(* IEC 61131-3 sources: greenbuddies-ems-concept/docs/data-model/codesys, 10 files *)

(* ---- EmsReference.st ---- *)
(* GENERATED by npm run model:generate. Create one DUT for each TYPE block. *)

TYPE ST_EmsMeta :
STRUCT
    Quality : USINT := 6; (* 0=good, 1=uncertain, 2=bad, 3=stale, 4=unsupported, 5=disabled, 6=initializing *)
    ObservedAtMs : ULINT; (* UTC Unix ms; 0 means unknown in this PLC adapter *)
    Sequence : UDINT; (* Per-point successful observation counter; wraps to 1 *)
END_STRUCT
END_TYPE

TYPE ST_EmsNumber :
STRUCT
    Value : LREAL;
    Meta : ST_EmsMeta;
END_STRUCT
END_TYPE

TYPE ST_EmsBoolean :
STRUCT
    Value : BOOL;
    Meta : ST_EmsMeta;
END_STRUCT
END_TYPE

TYPE ST_EmsText :
STRUCT
    Value : STRING(255);
    Meta : ST_EmsMeta;
END_STRUCT
END_TYPE

TYPE ST_EmsCounter :
STRUCT
    Value : ULINT;
    Meta : ST_EmsMeta;
END_STRUCT
END_TYPE

TYPE ST_EmsDecoded :
STRUCT
    Value : LREAL;
    Valid : BOOL;
END_STRUCT
END_TYPE

TYPE U_EmsReal32 :
UNION
    Bits : DWORD;
    Value : REAL;
END_UNION
END_TYPE

TYPE ST_EmsDevice :
STRUCT
    online : ST_EmsBoolean; (* device.online | state | r | Last device transaction succeeded; does not imply every point is healthy. *)
    state : ST_EmsText; (* device.state | state | r | Normalized operating state; unknown codes map to unknown, never running. *)
    available : ST_EmsBoolean; (* device.available | state | r | Device reports available for operation. *)
    remoteMode : ST_EmsBoolean; (* device.remoteMode | state | r | Device accepts remote control at its own interface. *)
    faultActive : ST_EmsBoolean; (* device.faultActive | state | r | At least one device fault is active. *)
    warningActive : ST_EmsBoolean; (* device.warningActive | state | r | At least one device warning is active. *)
    vendorCode : ST_EmsText; (* device.vendorCode | state | r | Unmodified diagnostic code for service; never drives portable UI behavior. *)
    latency : ST_EmsNumber; (* device.latency | ms | r | Most recent successful transaction duration. *)
    uptime : ST_EmsCounter; (* device.uptime | s | r | Device uptime. A reset is not negative consumption. *)
    communicationErrors : ST_EmsCounter; (* device.communicationErrors | count | r | Cumulative failed transactions since source restart. *)
END_STRUCT
END_TYPE

TYPE ST_EmsAc :
STRUCT
    activePower : ST_EmsNumber; (* ac.activePower | W | r | Signed active power at the declared measurement boundary. *)
    reactivePower : ST_EmsNumber; (* ac.reactivePower | var | r | Signed reactive power at the same boundary as activePower. *)
    apparentPower : ST_EmsNumber; (* ac.apparentPower | VA | r | Non-negative apparent power. *)
    frequency : ST_EmsNumber; (* ac.frequency | Hz | r | Measured AC frequency. *)
    powerFactor : ST_EmsNumber; (* ac.powerFactor | 1 | r | P / apparent power, signed by active power; null if undefined. *)
    voltageL1N : ST_EmsNumber; (* ac.voltageL1N | V | r | L1 to neutral RMS voltage. *)
    voltageL2N : ST_EmsNumber; (* ac.voltageL2N | V | r | L2 to neutral RMS voltage. *)
    voltageL3N : ST_EmsNumber; (* ac.voltageL3N | V | r | L3 to neutral RMS voltage. *)
    voltageL1L2 : ST_EmsNumber; (* ac.voltageL1L2 | V | r | L1 to L2 RMS voltage. *)
    voltageL2L3 : ST_EmsNumber; (* ac.voltageL2L3 | V | r | L2 to L3 RMS voltage. *)
    voltageL3L1 : ST_EmsNumber; (* ac.voltageL3L1 | V | r | L3 to L1 RMS voltage. *)
    currentL1 : ST_EmsNumber; (* ac.currentL1 | A | r | L1 RMS current magnitude. *)
    currentL2 : ST_EmsNumber; (* ac.currentL2 | A | r | L2 RMS current magnitude. *)
    currentL3 : ST_EmsNumber; (* ac.currentL3 | A | r | L3 RMS current magnitude. *)
    activePowerL1 : ST_EmsNumber; (* ac.activePowerL1 | W | r | Signed active power, L1. *)
    activePowerL2 : ST_EmsNumber; (* ac.activePowerL2 | W | r | Signed active power, L2. *)
    activePowerL3 : ST_EmsNumber; (* ac.activePowerL3 | W | r | Signed active power, L3. *)
    voltageThd : ST_EmsNumber; (* ac.voltageThd | % | r | Reported aggregate voltage total harmonic distortion. *)
END_STRUCT
END_TYPE

TYPE ST_EmsDc :
STRUCT
    voltage : ST_EmsNumber; (* dc.voltage | V | r | DC terminal voltage. *)
    current : ST_EmsNumber; (* dc.current | A | r | DC current; positive out of the asset. *)
    power : ST_EmsNumber; (* dc.power | W | r | DC power; positive out of the asset. *)
    insulationResistance : ST_EmsNumber; (* dc.insulationResistance | ohm | r | Insulation resistance to ground. *)
END_STRUCT
END_TYPE

TYPE ST_EmsEnergy :
STRUCT
    exported : ST_EmsCounter; (* energy.exported | Wh | r | Cumulative active energy leaving the boundary. *)
    imported : ST_EmsCounter; (* energy.imported | Wh | r | Cumulative active energy entering the boundary. *)
    generatedToday : ST_EmsNumber; (* energy.generatedToday | Wh | r | Generation since site-local midnight; date/timezone are metadata. *)
    exportedToday : ST_EmsNumber; (* energy.exportedToday | Wh | r | Export since site-local midnight. *)
    importedToday : ST_EmsNumber; (* energy.importedToday | Wh | r | Import since site-local midnight. *)
    runtime : ST_EmsCounter; (* energy.runtime | s | r | Cumulative operating time. *)
END_STRUCT
END_TYPE

TYPE ST_EmsPv :
STRUCT
    moduleTemperature : ST_EmsNumber; (* pv.moduleTemperature | degC | r | PV module temperature. *)
    inverterTemperature : ST_EmsNumber; (* pv.inverterTemperature | degC | r | Inverter internal temperature. *)
    irradiance : ST_EmsNumber; (* pv.irradiance | W/m2 | r | Plane-of-array irradiance. *)
    availablePower : ST_EmsNumber; (* pv.availablePower | W | r | Device-estimated available active power; not inferred from nameplate. *)
    curtailedPower : ST_EmsNumber; (* pv.curtailedPower | W | r | Reported curtailed active power. *)
END_STRUCT
END_TYPE

TYPE ST_EmsBattery :
STRUCT
    soc : ST_EmsNumber; (* battery.soc | % | r | State of charge. *)
    soh : ST_EmsNumber; (* battery.soh | % | r | State of health. *)
    storedEnergy : ST_EmsNumber; (* battery.storedEnergy | Wh | r | Estimated stored usable energy. *)
    chargeAvailable : ST_EmsNumber; (* battery.chargeAvailable | W | r | Maximum currently available charge magnitude. *)
    dischargeAvailable : ST_EmsNumber; (* battery.dischargeAvailable | W | r | Maximum currently available discharge magnitude. *)
    temperature : ST_EmsNumber; (* battery.temperature | degC | r | Reported representative battery temperature. *)
    minTemperature : ST_EmsNumber; (* battery.minTemperature | degC | r | Lowest measured temperature. *)
    maxTemperature : ST_EmsNumber; (* battery.maxTemperature | degC | r | Highest measured temperature. *)
    minCellVoltage : ST_EmsNumber; (* battery.minCellVoltage | V | r | Lowest measured cell voltage. *)
    maxCellVoltage : ST_EmsNumber; (* battery.maxCellVoltage | V | r | Highest measured cell voltage. *)
    cycles : ST_EmsCounter; (* battery.cycles | count | r | Completed equivalent cycles; fractional cycles require a separate extension field. *)
    contactorClosed : ST_EmsBoolean; (* battery.contactorClosed | state | r | Battery contactor closed readback. *)
    balancing : ST_EmsBoolean; (* battery.balancing | state | r | Cell balancing active. *)
END_STRUCT
END_TYPE

TYPE ST_EmsWind :
STRUCT
    speed : ST_EmsNumber; (* wind.speed | m/s | r | Wind speed at the instrument. *)
    direction : ST_EmsNumber; (* wind.direction | deg | r | Wind direction, clockwise from true north. *)
    rotorSpeed : ST_EmsNumber; (* wind.rotorSpeed | rpm | r | Rotor speed. *)
    nacelleDirection : ST_EmsNumber; (* wind.nacelleDirection | deg | r | Nacelle bearing from true north. *)
    pitch : ST_EmsNumber; (* wind.pitch | deg | r | Reported representative blade pitch. *)
    gearboxTemperature : ST_EmsNumber; (* wind.gearboxTemperature | degC | r | Gearbox temperature. *)
    availablePower : ST_EmsNumber; (* wind.availablePower | W | r | Reported available generation. *)
END_STRUCT
END_TYPE

TYPE ST_EmsHydro :
STRUCT
    flow : ST_EmsNumber; (* hydro.flow | m3/s | r | Volumetric flow through the unit. *)
    head : ST_EmsNumber; (* hydro.head | m | r | Net hydraulic head. *)
    upstreamLevel : ST_EmsNumber; (* hydro.upstreamLevel | m | r | Upstream level relative to the configured datum. *)
    downstreamLevel : ST_EmsNumber; (* hydro.downstreamLevel | m | r | Downstream level relative to the same datum. *)
    gatePosition : ST_EmsNumber; (* hydro.gatePosition | % | r | Gate opening. *)
    turbineSpeed : ST_EmsNumber; (* hydro.turbineSpeed | rpm | r | Hydro turbine speed. *)
    waterTemperature : ST_EmsNumber; (* hydro.waterTemperature | degC | r | Water temperature. *)
END_STRUCT
END_TYPE

TYPE ST_EmsGrid :
STRUCT
    dsoAllowance : ST_EmsNumber; (* grid.dsoAllowance | % | r | Discrete DSO export allowance. *)
    exportLimit : ST_EmsNumber; (* grid.exportLimit | W | r | Effective non-negative export ceiling. *)
    importLimit : ST_EmsNumber; (* grid.importLimit | W | r | Effective non-negative import ceiling. *)
    connected : ST_EmsBoolean; (* grid.connected | state | r | PCC connected to the external grid. *)
    islanded : ST_EmsBoolean; (* grid.islanded | state | r | Site operating as an island. *)
    breakerClosed : ST_EmsBoolean; (* grid.breakerClosed | state | r | Breaker closed auxiliary-contact readback. *)
    tripActive : ST_EmsBoolean; (* grid.tripActive | state | r | Protection trip active. *)
    transformerTemperature : ST_EmsNumber; (* grid.transformerTemperature | degC | r | Transformer winding or oil sensor, identified in point metadata. *)
    tapPosition : ST_EmsNumber; (* grid.tapPosition | step | r | Transformer tap position; signed integral step. *)
END_STRUCT
END_TYPE

TYPE ST_EmsMeteo :
STRUCT
    airTemperature : ST_EmsNumber; (* meteo.airTemperature | degC | r | Ambient air temperature. *)
    humidity : ST_EmsNumber; (* meteo.humidity | % | r | Relative humidity. *)
    pressure : ST_EmsNumber; (* meteo.pressure | Pa | r | Atmospheric pressure. *)
    irradiance : ST_EmsNumber; (* meteo.irradiance | W/m2 | r | Global horizontal irradiance. *)
    windSpeed : ST_EmsNumber; (* meteo.windSpeed | m/s | r | Wind speed. *)
    windDirection : ST_EmsNumber; (* meteo.windDirection | deg | r | Direction clockwise from true north. *)
    rainfall : ST_EmsNumber; (* meteo.rainfall | mm | r | Precipitation in the configured measurement window. *)
END_STRUCT
END_TYPE

TYPE ST_EmsLoad :
STRUCT
    demand : ST_EmsNumber; (* load.demand | W | r | Non-negative active power consumed. *)
    flexiblePower : ST_EmsNumber; (* load.flexiblePower | W | r | Reported shed-able load magnitude. *)
    enabled : ST_EmsBoolean; (* load.enabled | state | r | Load enabled readback. *)
    vehicleConnected : ST_EmsBoolean; (* load.vehicleConnected | state | r | Vehicle present at this connector. *)
    charging : ST_EmsBoolean; (* load.charging | state | r | Charging active readback. *)
    currentLimit : ST_EmsNumber; (* load.currentLimit | A | r | Accepted EV connector current limit. *)
    sessionEnergy : ST_EmsNumber; (* load.sessionEnergy | Wh | r | Energy delivered in this charging session. *)
END_STRUCT
END_TYPE

TYPE ST_EmsController :
STRUCT
    mode : ST_EmsText; (* controller.mode | state | r | Current controller mode. *)
    source : ST_EmsText; (* controller.source | state | r | Exactly one selected command authority. *)
    remoteConnected : ST_EmsBoolean; (* controller.remoteConnected | state | r | Aggregator transport connected. *)
    remoteAllowed : ST_EmsBoolean; (* controller.remoteAllowed | state | rw | Remote permission readback; disabling selects local authority. *)
    requestedPower : ST_EmsNumber; (* controller.requestedPower | W | r | Requested aggregate active power before controller constraints. *)
    afterController : ST_EmsNumber; (* controller.afterController | W | r | Power after local optimization and device feasibility limits. *)
    afterDso : ST_EmsNumber; (* controller.afterDso | W | r | Power after DSO/export constraints. *)
    deliveredPower : ST_EmsNumber; (* controller.deliveredPower | W | r | Final dispatched power; distinct from measured power. *)
    limitingReason : ST_EmsText; (* controller.limitingReason | state | r | Dominant normalized active constraint. *)
END_STRUCT
END_TYPE

TYPE ST_EmsSettings :
STRUCT
    peakImportTarget : ST_EmsNumber; (* settings.peakImportTarget | W | rw | Peak-shaving import target. *)
    peakShavingShare : ST_EmsNumber; (* settings.peakShavingShare | % | rw | Usable battery allocation to peak shaving; remainder for load shifting. *)
    socMin : ST_EmsNumber; (* settings.socMin | % | rw | Minimum operating SoC; strictly below socMax. *)
    socMax : ST_EmsNumber; (* settings.socMax | % | rw | Maximum operating SoC; strictly above socMin. *)
    chargeLimit : ST_EmsNumber; (* settings.chargeLimit | W | rw | Requested maximum charge magnitude. *)
    dischargeLimit : ST_EmsNumber; (* settings.dischargeLimit | W | rw | Requested maximum discharge magnitude. *)
    rampLimit : ST_EmsNumber; (* settings.rampLimit | W/s | rw | Maximum change of active power magnitude per second. *)
END_STRUCT
END_TYPE

TYPE ST_EmsCamera :
STRUCT
    online : ST_EmsBoolean; (* camera.online | state | r | Camera reachable. *)
    recording : ST_EmsBoolean; (* camera.recording | state | r | Recording active. *)
    frameAge : ST_EmsNumber; (* camera.frameAge | ms | r | Age of most recently received image. *)
END_STRUCT
END_TYPE

TYPE ST_EmsAsset :
STRUCT
    Id : STRING(128);
    Kind : STRING(32);
    device : ST_EmsDevice;
    ac : ST_EmsAc;
    dc : ST_EmsDc;
    energy : ST_EmsEnergy;
    pv : ST_EmsPv;
    battery : ST_EmsBattery;
    wind : ST_EmsWind;
    hydro : ST_EmsHydro;
    grid : ST_EmsGrid;
    meteo : ST_EmsMeteo;
    load : ST_EmsLoad;
    controller : ST_EmsController;
    settings : ST_EmsSettings;
    camera : ST_EmsCamera;
END_STRUCT
END_TYPE

(* Additional DUTs. Fixed reference bounds: 64 intervals, 32 targets per interval. Reject larger input before copying. *)
TYPE ST_EmsTarget :
STRUCT
    AssetId : STRING(128);
    ActivePowerW : LREAL;
END_STRUCT
END_TYPE

TYPE ST_EmsInterval :
STRUCT
    StartMs : ULINT;
    EndMs : ULINT;
    TargetCount : UINT;
    Targets : ARRAY[1..32] OF ST_EmsTarget;
END_STRUCT
END_TYPE

TYPE ST_EmsProfile :
STRUCT
    Revision : STRING(128);
    ValidFromMs : ULINT;
    ValidUntilMs : ULINT;
    IntervalCount : UINT;
    Intervals : ARRAY[1..64] OF ST_EmsInterval;
END_STRUCT
END_TYPE

TYPE ST_EmsCommandResult :
STRUCT
    CommandId : STRING(128);
    Revision : STRING(128);
    State : STRING(32); (* received, validated, accepted, applied, rejected, expired *)
    Reason : STRING(255);
    AtMs : ULINT;
END_STRUCT
END_TYPE

(* ===== FB_EmsHighAlarm.st ===== *)
(* Create a FUNCTION_BLOCK POU. Declarations above, implementation below the divider.
   Requires the CODESYS Standard library (TON). Example settings are not safety limits.
   One instance per condition. Call every scan from ONE acquisition/alarm task.
   Acknowledgement belongs to Alarm Manager, never to this block. *)
FUNCTION_BLOCK FB_EmsHighAlarm
VAR_INPUT
    lrValue       : LREAL;
    xValid        : BOOL;        (* Good, fresh sample AND valid mapping *)
    lrHigh        : LREAL;
    lrReset       : LREAL;       (* Must be below lrHigh: hysteresis *)
    tRaiseDelay   : TIME := T#2s;
    tClearDelay   : TIME := T#5s;
END_VAR
VAR_OUTPUT
    xActive       : BOOL;        (* Digital alarm expression; never writable by HMI *)
    xInputFault   : BOOL;        (* Separate communication/measurement alarm *)
    xConfigFault  : BOOL;
END_VAR
VAR
    fbRaise       : TON;
    fbClear       : TON;
END_VAR
(* ---- Implementation ---- *)
xConfigFault := (lrReset >= lrHigh);
xInputFault := NOT xValid;
IF xInputFault OR xConfigFault THEN
    fbRaise(IN := FALSE, PT := tRaiseDelay);
    fbClear(IN := FALSE, PT := tClearDelay);
    (* Hold last known condition; unavailable data must not clear a fault. *)
ELSE
    fbRaise(IN := (NOT xActive) AND (lrValue >= lrHigh), PT := tRaiseDelay);
    fbClear(IN := xActive AND (lrValue <= lrReset), PT := tClearDelay);
    IF fbRaise.Q THEN
        xActive := TRUE;
    ELSIF fbClear.Q THEN
        xActive := FALSE;
    END_IF;
END_IF;
END_FUNCTION_BLOCK

(* ===== FB_EmsSample.st ===== *)
(* POU: FUNCTION_BLOCK FB_EmsSample. Declaration above the divider; implementation below it. *)
FUNCTION_BLOCK FB_EmsSample
VAR_INPUT
    xSupported : BOOL := TRUE;
    xEnabled : BOOL := TRUE;
    xNewSample : BOOL; (* One pulse per completed acquisition, NOT each PLC cycle. *)
    xReadError : BOOL; (* Failed transaction pulse; retained words are not new data. *)
    xValueValid : BOOL := TRUE;
    xClockValid : BOOL;
    uliUtcMs : ULINT;
    uliMonotonicMs : ULINT; (* LTIME_TO_ULINT(LTIME()) / ULINT#1000000 *)
    udiStaleAfterMs : UDINT := 5000;
END_VAR
VAR_OUTPUT
    Meta : ST_EmsMeta;
    xAccept : BOOL; (* Copy the decoded value only when TRUE. *)
END_VAR
VAR
    xSeen : BOOL;
    uliLastMs : ULINT;
END_VAR
(* IMPLEMENTATION *)
xAccept := FALSE;
IF NOT xSupported THEN
    Meta.Quality := 4; (* unsupported *)
    Meta.ObservedAtMs := 0;
    Meta.Sequence := 0;
    xSeen := FALSE;
ELSIF NOT xEnabled THEN
    Meta.Quality := 5; (* disabled; retain the last observation *)
ELSIF xReadError THEN
    Meta.Quality := 2; (* bad; preserve last observation time and value *)
ELSIF xNewSample THEN
    IF xValueValid THEN
        xAccept := TRUE;
        xSeen := TRUE;
        uliLastMs := uliMonotonicMs;
        IF xClockValid AND (uliUtcMs > 0) THEN
            Meta.Quality := 0;
            Meta.ObservedAtMs := uliUtcMs;
        ELSE
            Meta.Quality := 1; (* uncertain: no trustworthy UTC *)
            Meta.ObservedAtMs := 0;
        END_IF;
        IF Meta.Sequence = UDINT#4294967295 THEN
            Meta.Sequence := 1;
        ELSE
            Meta.Sequence := Meta.Sequence + 1;
        END_IF;
    ELSE
        Meta.Quality := 2; (* sentinel, range error or unmapped enum *)
    END_IF;
ELSIF xSeen THEN
    IF uliMonotonicMs < uliLastMs THEN
        Meta.Quality := 2; (* monotonic clock reset; wait for a new sample *)
    ELSIF (uliMonotonicMs - uliLastMs) > UDINT_TO_ULINT(udiStaleAfterMs) THEN
        Meta.Quality := 3; (* stale; UTC observation time stays unchanged *)
    END_IF;
END_IF;
END_FUNCTION_BLOCK

(* ===== F_EmsDecode32.st ===== *)
(* POU: FUNCTION F_EmsDecode32. Raw words from ONE successful Modbus transaction. *)
FUNCTION F_EmsDecode32 : ST_EmsDecoded
VAR_INPUT
    wFirst : WORD;
    wSecond : WORD;
    xLowWordFirst : BOOL;
    xLowByteFirst : BOOL;
    usiEncoding : USINT; (* 0=uint16, 1=int16, 2=uint32, 3=int32, 4=float32 *)
    lrScale : LREAL := 1;
    lrOffset : LREAL;
    xHasSentinel : BOOL;
    dwSentinel : DWORD; (* Canonical bit order BEFORE scaling *)
END_VAR
VAR
    wA, wB, wTemporary : WORD;
    dwBits : DWORD;
    uBits : U_EmsReal32;
    lrRaw : LREAL;
END_VAR
(* IMPLEMENTATION *)
F_EmsDecode32.Valid := FALSE;
F_EmsDecode32.Value := 0;
wA := wFirst;
wB := wSecond;
IF xLowByteFirst THEN
    wA := SHL(wA AND WORD#16#00FF, 8) OR SHR(wA, 8);
    wB := SHL(wB AND WORD#16#00FF, 8) OR SHR(wB, 8);
END_IF;
IF xLowWordFirst AND (usiEncoding >= 2) THEN
    wTemporary := wA; wA := wB; wB := wTemporary;
END_IF;
IF usiEncoding < 2 THEN
    dwBits := WORD_TO_DWORD(wA);
ELSE
    dwBits := SHL(WORD_TO_DWORD(wA), 16) OR WORD_TO_DWORD(wB);
END_IF;
IF xHasSentinel AND (dwBits = dwSentinel) THEN RETURN; END_IF;
CASE usiEncoding OF
    0: lrRaw := WORD_TO_LREAL(wA);
    1:
        lrRaw := WORD_TO_LREAL(wA);
        IF wA >= WORD#16#8000 THEN lrRaw := lrRaw - LREAL#65536; END_IF;
    2: lrRaw := UDINT_TO_LREAL(DWORD_TO_UDINT(dwBits));
    3:
        lrRaw := UDINT_TO_LREAL(DWORD_TO_UDINT(dwBits));
        IF dwBits >= DWORD#16#80000000 THEN lrRaw := lrRaw - LREAL#4294967296; END_IF;
    4:
        IF (dwBits AND DWORD#16#7F800000) = DWORD#16#7F800000 THEN RETURN; END_IF; (* NaN/Inf *)
        uBits.Bits := dwBits;
        lrRaw := REAL_TO_LREAL(uBits.Value);
ELSE
    RETURN;
END_CASE;
F_EmsDecode32.Value := lrRaw * lrScale + lrOffset;
(* Practical engineering bound rejects NaN/overflow without target-specific math libraries. *)
F_EmsDecode32.Valid := (F_EmsDecode32.Value = F_EmsDecode32.Value)
    AND (ABS(F_EmsDecode32.Value) <= LREAL#1.0E30) AND (lrScale <> 0);
END_FUNCTION

(* ===== F_EmsDecode64.st ===== *)
(* POU: FUNCTION F_EmsDecode64. Exact UInt64 reconstruction; never pass via LREAL. *)
FUNCTION F_EmsDecode64 : ULINT
VAR_INPUT
    Words : ARRAY[0..3] OF WORD;
    xLowWordFirst : BOOL;
    xLowByteFirst : BOOL;
END_VAR
VAR
    i, j : INT;
    w : WORD;
END_VAR
(* IMPLEMENTATION *)
F_EmsDecode64 := 0;
FOR i := 0 TO 3 DO
    IF xLowWordFirst THEN j := 3 - i; ELSE j := i; END_IF;
    w := Words[j];
    IF xLowByteFirst THEN
        w := SHL(w AND WORD#16#00FF, 8) OR SHR(w, 8);
    END_IF;
    F_EmsDecode64 := SHL(F_EmsDecode64, 16) OR WORD_TO_ULINT(w);
END_FOR;
(* Validate the vendor's invalid sentinel before passing xValueValid to FB_EmsSample. *)
END_FUNCTION

(* ===== GVL_Ems.st ===== *)
(* Global Variable List named GVL_Ems. Export read-only; do not mark this GVL RETAIN. *)
{attribute 'qualified_only'}
VAR_GLOBAL
    Battery : ST_EmsAsset := (Id := 'BESS-01', Kind := 'battery-system');
END_VAR

(* ===== PRG_EmsAlarms.st ===== *)
(* Reference only: wire these inputs to the completed Modbus acquisition result.
   xTemperatureValid must include freshness, device health, range and finite-value checks.
   Schedule this program cyclically. Choose limits/delays during commissioning. *)
PROGRAM PRG_EmsAlarms
VAR
    lrTemperatureC    : LREAL;
    xTemperatureValid: BOOL := FALSE;
    fbTemperature    : FB_EmsHighAlarm;
END_VAR
(* ---- Implementation ---- *)
fbTemperature(
    lrValue := lrTemperatureC,
    xValid := xTemperatureValid,
    lrHigh := 45.0,
    lrReset := 42.0,
    tRaiseDelay := T#2s,
    tClearDelay := T#5s
);
(* Alarm Manager / digital expressions:
   bess.temperature.high    := PRG_EmsAlarms.fbTemperature.xActive
   bess.temperature.invalid := PRG_EmsAlarms.fbTemperature.xInputFault
   bess.alarm.config        := PRG_EmsAlarms.fbTemperature.xConfigFault
   Define all three in an ACK_REP alarm class. Do not reset digital alarms on ACK.
   Alarm Manager owns occurrence state, timestamps, archive and acknowledgment.
   These expressions do NOT need individual OPC UA boolean tag subscriptions. *)
END_PROGRAM

(* ===== PRG_EmsExample.st ===== *)
(* POU: PROGRAM PRG_EmsExample. Map the Inputs through your completed Modbus request. *)
PROGRAM PRG_EmsExample
VAR
    (* Replace these driver-bound inputs; none are invented automatic CODESYS diagnostics. *)
    aBatteryWords : ARRAY[0..2] OF WORD;
    xBatteryDone : BOOL; (* one pulse for a successful complete response *)
    xBatteryError : BOOL;
    xUtcSynchronized : BOOL;
    uliUtcMs : ULINT; (* Fill from SysTimeRtcHighResGet + clock synchronization health. *)
    uliMonotonicMs : ULINT;
    powerSample : FB_EmsSample;
    socSample : FB_EmsSample;
    decoded : ST_EmsDecoded;
    lrSoc : LREAL;
END_VAR
(* IMPLEMENTATION *)
uliMonotonicMs := LTIME_TO_ULINT(LTIME()) / ULINT#1000000;
(* Example vendor: signed kW, positive charge. Convert ONCE to W, positive discharge. *)
decoded := F_EmsDecode32(wFirst := aBatteryWords[0], wSecond := aBatteryWords[1],
    xLowWordFirst := FALSE, xLowByteFirst := FALSE, usiEncoding := 3,
    lrScale := -1000, lrOffset := 0, xHasSentinel := TRUE, dwSentinel := DWORD#16#80000000);
powerSample(xNewSample := xBatteryDone, xReadError := xBatteryError,
    xValueValid := decoded.Valid AND (ABS(decoded.Value) <= LREAL#2000000),
    xClockValid := xUtcSynchronized, uliUtcMs := uliUtcMs,
    uliMonotonicMs := uliMonotonicMs, udiStaleAfterMs := 5000);
IF powerSample.xAccept THEN GVL_Ems.Battery.ac.activePower.Value := decoded.Value; END_IF;
GVL_Ems.Battery.ac.activePower.Meta := powerSample.Meta;

lrSoc := WORD_TO_LREAL(aBatteryWords[2]) * LREAL#0.1;
socSample(xNewSample := xBatteryDone, xReadError := xBatteryError,
    xValueValid := (aBatteryWords[2] <> WORD#16#FFFF) AND (lrSoc >= 0) AND (lrSoc <= 100),
    xClockValid := xUtcSynchronized, uliUtcMs := uliUtcMs,
    uliMonotonicMs := uliMonotonicMs, udiStaleAfterMs := 5000);
IF socSample.xAccept THEN GVL_Ems.Battery.battery.soc.Value := lrSoc; END_IF;
GVL_Ems.Battery.battery.soc.Meta := socSample.Meta;
(* Call in one acquisition task. Do not expose a partially updated struct as an atomic snapshot. *)
END_PROGRAM

(* ---- ProfileTypes.st ---- *)
(* Additional DUTs. Fixed reference bounds: 64 intervals, 32 targets per interval. Reject larger input before copying. *)
TYPE ST_EmsTarget :
STRUCT
    AssetId : STRING(128);
    ActivePowerW : LREAL;
END_STRUCT
END_TYPE

TYPE ST_EmsInterval :
STRUCT
    StartMs : ULINT;
    EndMs : ULINT;
    TargetCount : UINT;
    Targets : ARRAY[1..32] OF ST_EmsTarget;
END_STRUCT
END_TYPE

TYPE ST_EmsProfile :
STRUCT
    Revision : STRING(128);
    ValidFromMs : ULINT;
    ValidUntilMs : ULINT;
    IntervalCount : UINT;
    Intervals : ARRAY[1..64] OF ST_EmsInterval;
END_STRUCT
END_TYPE

TYPE ST_EmsCommandResult :
STRUCT
    CommandId : STRING(128);
    Revision : STRING(128);
    State : STRING(32); (* received, validated, accepted, applied, rejected, expired *)
    Reason : STRING(255);
    AtMs : ULINT;
END_STRUCT
END_TYPE

(* ---- Types.st ---- *)
(* GENERATED by npm run model:generate. Create one DUT for each TYPE block. *)

TYPE ST_EmsMeta :
STRUCT
    Quality : USINT := 6; (* 0=good, 1=uncertain, 2=bad, 3=stale, 4=unsupported, 5=disabled, 6=initializing *)
    ObservedAtMs : ULINT; (* UTC Unix ms; 0 means unknown in this PLC adapter *)
    Sequence : UDINT; (* Per-point successful observation counter; wraps to 1 *)
END_STRUCT
END_TYPE

TYPE ST_EmsNumber :
STRUCT
    Value : LREAL;
    Meta : ST_EmsMeta;
END_STRUCT
END_TYPE

TYPE ST_EmsBoolean :
STRUCT
    Value : BOOL;
    Meta : ST_EmsMeta;
END_STRUCT
END_TYPE

TYPE ST_EmsText :
STRUCT
    Value : STRING(255);
    Meta : ST_EmsMeta;
END_STRUCT
END_TYPE

TYPE ST_EmsCounter :
STRUCT
    Value : ULINT;
    Meta : ST_EmsMeta;
END_STRUCT
END_TYPE

TYPE ST_EmsDecoded :
STRUCT
    Value : LREAL;
    Valid : BOOL;
END_STRUCT
END_TYPE

TYPE U_EmsReal32 :
UNION
    Bits : DWORD;
    Value : REAL;
END_UNION
END_TYPE

TYPE ST_EmsDevice :
STRUCT
    online : ST_EmsBoolean; (* device.online | state | r | Last device transaction succeeded; does not imply every point is healthy. *)
    state : ST_EmsText; (* device.state | state | r | Normalized operating state; unknown codes map to unknown, never running. *)
    available : ST_EmsBoolean; (* device.available | state | r | Device reports available for operation. *)
    remoteMode : ST_EmsBoolean; (* device.remoteMode | state | r | Device accepts remote control at its own interface. *)
    faultActive : ST_EmsBoolean; (* device.faultActive | state | r | At least one device fault is active. *)
    warningActive : ST_EmsBoolean; (* device.warningActive | state | r | At least one device warning is active. *)
    vendorCode : ST_EmsText; (* device.vendorCode | state | r | Unmodified diagnostic code for service; never drives portable UI behavior. *)
    latency : ST_EmsNumber; (* device.latency | ms | r | Most recent successful transaction duration. *)
    uptime : ST_EmsCounter; (* device.uptime | s | r | Device uptime. A reset is not negative consumption. *)
    communicationErrors : ST_EmsCounter; (* device.communicationErrors | count | r | Cumulative failed transactions since source restart. *)
END_STRUCT
END_TYPE

TYPE ST_EmsAc :
STRUCT
    activePower : ST_EmsNumber; (* ac.activePower | W | r | Signed active power at the declared measurement boundary. *)
    reactivePower : ST_EmsNumber; (* ac.reactivePower | var | r | Signed reactive power at the same boundary as activePower. *)
    apparentPower : ST_EmsNumber; (* ac.apparentPower | VA | r | Non-negative apparent power. *)
    frequency : ST_EmsNumber; (* ac.frequency | Hz | r | Measured AC frequency. *)
    powerFactor : ST_EmsNumber; (* ac.powerFactor | 1 | r | P / apparent power, signed by active power; null if undefined. *)
    voltageL1N : ST_EmsNumber; (* ac.voltageL1N | V | r | L1 to neutral RMS voltage. *)
    voltageL2N : ST_EmsNumber; (* ac.voltageL2N | V | r | L2 to neutral RMS voltage. *)
    voltageL3N : ST_EmsNumber; (* ac.voltageL3N | V | r | L3 to neutral RMS voltage. *)
    voltageL1L2 : ST_EmsNumber; (* ac.voltageL1L2 | V | r | L1 to L2 RMS voltage. *)
    voltageL2L3 : ST_EmsNumber; (* ac.voltageL2L3 | V | r | L2 to L3 RMS voltage. *)
    voltageL3L1 : ST_EmsNumber; (* ac.voltageL3L1 | V | r | L3 to L1 RMS voltage. *)
    currentL1 : ST_EmsNumber; (* ac.currentL1 | A | r | L1 RMS current magnitude. *)
    currentL2 : ST_EmsNumber; (* ac.currentL2 | A | r | L2 RMS current magnitude. *)
    currentL3 : ST_EmsNumber; (* ac.currentL3 | A | r | L3 RMS current magnitude. *)
    activePowerL1 : ST_EmsNumber; (* ac.activePowerL1 | W | r | Signed active power, L1. *)
    activePowerL2 : ST_EmsNumber; (* ac.activePowerL2 | W | r | Signed active power, L2. *)
    activePowerL3 : ST_EmsNumber; (* ac.activePowerL3 | W | r | Signed active power, L3. *)
    voltageThd : ST_EmsNumber; (* ac.voltageThd | % | r | Reported aggregate voltage total harmonic distortion. *)
END_STRUCT
END_TYPE

TYPE ST_EmsDc :
STRUCT
    voltage : ST_EmsNumber; (* dc.voltage | V | r | DC terminal voltage. *)
    current : ST_EmsNumber; (* dc.current | A | r | DC current; positive out of the asset. *)
    power : ST_EmsNumber; (* dc.power | W | r | DC power; positive out of the asset. *)
    insulationResistance : ST_EmsNumber; (* dc.insulationResistance | ohm | r | Insulation resistance to ground. *)
END_STRUCT
END_TYPE

TYPE ST_EmsEnergy :
STRUCT
    exported : ST_EmsCounter; (* energy.exported | Wh | r | Cumulative active energy leaving the boundary. *)
    imported : ST_EmsCounter; (* energy.imported | Wh | r | Cumulative active energy entering the boundary. *)
    generatedToday : ST_EmsNumber; (* energy.generatedToday | Wh | r | Generation since site-local midnight; date/timezone are metadata. *)
    exportedToday : ST_EmsNumber; (* energy.exportedToday | Wh | r | Export since site-local midnight. *)
    importedToday : ST_EmsNumber; (* energy.importedToday | Wh | r | Import since site-local midnight. *)
    runtime : ST_EmsCounter; (* energy.runtime | s | r | Cumulative operating time. *)
END_STRUCT
END_TYPE

TYPE ST_EmsPv :
STRUCT
    moduleTemperature : ST_EmsNumber; (* pv.moduleTemperature | degC | r | PV module temperature. *)
    inverterTemperature : ST_EmsNumber; (* pv.inverterTemperature | degC | r | Inverter internal temperature. *)
    irradiance : ST_EmsNumber; (* pv.irradiance | W/m2 | r | Plane-of-array irradiance. *)
    availablePower : ST_EmsNumber; (* pv.availablePower | W | r | Device-estimated available active power; not inferred from nameplate. *)
    curtailedPower : ST_EmsNumber; (* pv.curtailedPower | W | r | Reported curtailed active power. *)
END_STRUCT
END_TYPE

TYPE ST_EmsBattery :
STRUCT
    soc : ST_EmsNumber; (* battery.soc | % | r | State of charge. *)
    soh : ST_EmsNumber; (* battery.soh | % | r | State of health. *)
    storedEnergy : ST_EmsNumber; (* battery.storedEnergy | Wh | r | Estimated stored usable energy. *)
    chargeAvailable : ST_EmsNumber; (* battery.chargeAvailable | W | r | Maximum currently available charge magnitude. *)
    dischargeAvailable : ST_EmsNumber; (* battery.dischargeAvailable | W | r | Maximum currently available discharge magnitude. *)
    temperature : ST_EmsNumber; (* battery.temperature | degC | r | Reported representative battery temperature. *)
    minTemperature : ST_EmsNumber; (* battery.minTemperature | degC | r | Lowest measured temperature. *)
    maxTemperature : ST_EmsNumber; (* battery.maxTemperature | degC | r | Highest measured temperature. *)
    minCellVoltage : ST_EmsNumber; (* battery.minCellVoltage | V | r | Lowest measured cell voltage. *)
    maxCellVoltage : ST_EmsNumber; (* battery.maxCellVoltage | V | r | Highest measured cell voltage. *)
    cycles : ST_EmsCounter; (* battery.cycles | count | r | Completed equivalent cycles; fractional cycles require a separate extension field. *)
    contactorClosed : ST_EmsBoolean; (* battery.contactorClosed | state | r | Battery contactor closed readback. *)
    balancing : ST_EmsBoolean; (* battery.balancing | state | r | Cell balancing active. *)
END_STRUCT
END_TYPE

TYPE ST_EmsWind :
STRUCT
    speed : ST_EmsNumber; (* wind.speed | m/s | r | Wind speed at the instrument. *)
    direction : ST_EmsNumber; (* wind.direction | deg | r | Wind direction, clockwise from true north. *)
    rotorSpeed : ST_EmsNumber; (* wind.rotorSpeed | rpm | r | Rotor speed. *)
    nacelleDirection : ST_EmsNumber; (* wind.nacelleDirection | deg | r | Nacelle bearing from true north. *)
    pitch : ST_EmsNumber; (* wind.pitch | deg | r | Reported representative blade pitch. *)
    gearboxTemperature : ST_EmsNumber; (* wind.gearboxTemperature | degC | r | Gearbox temperature. *)
    availablePower : ST_EmsNumber; (* wind.availablePower | W | r | Reported available generation. *)
END_STRUCT
END_TYPE

TYPE ST_EmsHydro :
STRUCT
    flow : ST_EmsNumber; (* hydro.flow | m3/s | r | Volumetric flow through the unit. *)
    head : ST_EmsNumber; (* hydro.head | m | r | Net hydraulic head. *)
    upstreamLevel : ST_EmsNumber; (* hydro.upstreamLevel | m | r | Upstream level relative to the configured datum. *)
    downstreamLevel : ST_EmsNumber; (* hydro.downstreamLevel | m | r | Downstream level relative to the same datum. *)
    gatePosition : ST_EmsNumber; (* hydro.gatePosition | % | r | Gate opening. *)
    turbineSpeed : ST_EmsNumber; (* hydro.turbineSpeed | rpm | r | Hydro turbine speed. *)
    waterTemperature : ST_EmsNumber; (* hydro.waterTemperature | degC | r | Water temperature. *)
END_STRUCT
END_TYPE

TYPE ST_EmsGrid :
STRUCT
    dsoAllowance : ST_EmsNumber; (* grid.dsoAllowance | % | r | Discrete DSO export allowance. *)
    exportLimit : ST_EmsNumber; (* grid.exportLimit | W | r | Effective non-negative export ceiling. *)
    importLimit : ST_EmsNumber; (* grid.importLimit | W | r | Effective non-negative import ceiling. *)
    connected : ST_EmsBoolean; (* grid.connected | state | r | PCC connected to the external grid. *)
    islanded : ST_EmsBoolean; (* grid.islanded | state | r | Site operating as an island. *)
    breakerClosed : ST_EmsBoolean; (* grid.breakerClosed | state | r | Breaker closed auxiliary-contact readback. *)
    tripActive : ST_EmsBoolean; (* grid.tripActive | state | r | Protection trip active. *)
    transformerTemperature : ST_EmsNumber; (* grid.transformerTemperature | degC | r | Transformer winding or oil sensor, identified in point metadata. *)
    tapPosition : ST_EmsNumber; (* grid.tapPosition | step | r | Transformer tap position; signed integral step. *)
END_STRUCT
END_TYPE

TYPE ST_EmsMeteo :
STRUCT
    airTemperature : ST_EmsNumber; (* meteo.airTemperature | degC | r | Ambient air temperature. *)
    humidity : ST_EmsNumber; (* meteo.humidity | % | r | Relative humidity. *)
    pressure : ST_EmsNumber; (* meteo.pressure | Pa | r | Atmospheric pressure. *)
    irradiance : ST_EmsNumber; (* meteo.irradiance | W/m2 | r | Global horizontal irradiance. *)
    windSpeed : ST_EmsNumber; (* meteo.windSpeed | m/s | r | Wind speed. *)
    windDirection : ST_EmsNumber; (* meteo.windDirection | deg | r | Direction clockwise from true north. *)
    rainfall : ST_EmsNumber; (* meteo.rainfall | mm | r | Precipitation in the configured measurement window. *)
END_STRUCT
END_TYPE

TYPE ST_EmsLoad :
STRUCT
    demand : ST_EmsNumber; (* load.demand | W | r | Non-negative active power consumed. *)
    flexiblePower : ST_EmsNumber; (* load.flexiblePower | W | r | Reported shed-able load magnitude. *)
    enabled : ST_EmsBoolean; (* load.enabled | state | r | Load enabled readback. *)
    vehicleConnected : ST_EmsBoolean; (* load.vehicleConnected | state | r | Vehicle present at this connector. *)
    charging : ST_EmsBoolean; (* load.charging | state | r | Charging active readback. *)
    currentLimit : ST_EmsNumber; (* load.currentLimit | A | r | Accepted EV connector current limit. *)
    sessionEnergy : ST_EmsNumber; (* load.sessionEnergy | Wh | r | Energy delivered in this charging session. *)
END_STRUCT
END_TYPE

TYPE ST_EmsController :
STRUCT
    mode : ST_EmsText; (* controller.mode | state | r | Current controller mode. *)
    source : ST_EmsText; (* controller.source | state | r | Exactly one selected command authority. *)
    remoteConnected : ST_EmsBoolean; (* controller.remoteConnected | state | r | Aggregator transport connected. *)
    remoteAllowed : ST_EmsBoolean; (* controller.remoteAllowed | state | rw | Remote permission readback; disabling selects local authority. *)
    requestedPower : ST_EmsNumber; (* controller.requestedPower | W | r | Requested aggregate active power before controller constraints. *)
    afterController : ST_EmsNumber; (* controller.afterController | W | r | Power after local optimization and device feasibility limits. *)
    afterDso : ST_EmsNumber; (* controller.afterDso | W | r | Power after DSO/export constraints. *)
    deliveredPower : ST_EmsNumber; (* controller.deliveredPower | W | r | Final dispatched power; distinct from measured power. *)
    limitingReason : ST_EmsText; (* controller.limitingReason | state | r | Dominant normalized active constraint. *)
END_STRUCT
END_TYPE

TYPE ST_EmsSettings :
STRUCT
    peakImportTarget : ST_EmsNumber; (* settings.peakImportTarget | W | rw | Peak-shaving import target. *)
    peakShavingShare : ST_EmsNumber; (* settings.peakShavingShare | % | rw | Usable battery allocation to peak shaving; remainder for load shifting. *)
    socMin : ST_EmsNumber; (* settings.socMin | % | rw | Minimum operating SoC; strictly below socMax. *)
    socMax : ST_EmsNumber; (* settings.socMax | % | rw | Maximum operating SoC; strictly above socMin. *)
    chargeLimit : ST_EmsNumber; (* settings.chargeLimit | W | rw | Requested maximum charge magnitude. *)
    dischargeLimit : ST_EmsNumber; (* settings.dischargeLimit | W | rw | Requested maximum discharge magnitude. *)
    rampLimit : ST_EmsNumber; (* settings.rampLimit | W/s | rw | Maximum change of active power magnitude per second. *)
END_STRUCT
END_TYPE

TYPE ST_EmsCamera :
STRUCT
    online : ST_EmsBoolean; (* camera.online | state | r | Camera reachable. *)
    recording : ST_EmsBoolean; (* camera.recording | state | r | Recording active. *)
    frameAge : ST_EmsNumber; (* camera.frameAge | ms | r | Age of most recently received image. *)
END_STRUCT
END_TYPE

TYPE ST_EmsAsset :
STRUCT
    Id : STRING(128);
    Kind : STRING(32);
    device : ST_EmsDevice;
    ac : ST_EmsAc;
    dc : ST_EmsDc;
    energy : ST_EmsEnergy;
    pv : ST_EmsPv;
    battery : ST_EmsBattery;
    wind : ST_EmsWind;
    hydro : ST_EmsHydro;
    grid : ST_EmsGrid;
    meteo : ST_EmsMeteo;
    load : ST_EmsLoad;
    controller : ST_EmsController;
    settings : ST_EmsSettings;
    camera : ST_EmsCamera;
END_STRUCT
END_TYPE

(* ---- GVL_Ems.st ---- *)
(* Global Variable List named GVL_Ems. Export read-only; do not mark this GVL RETAIN. *)
{attribute 'qualified_only'}
VAR_GLOBAL
    Battery : ST_EmsAsset := (Id := 'BESS-01', Kind := 'battery-system');
END_VAR

(* ---- F_EmsDecode32.st ---- *)
(* POU: FUNCTION F_EmsDecode32. Raw words from ONE successful Modbus transaction. *)
FUNCTION F_EmsDecode32 : ST_EmsDecoded
VAR_INPUT
    wFirst : WORD;
    wSecond : WORD;
    xLowWordFirst : BOOL;
    xLowByteFirst : BOOL;
    usiEncoding : USINT; (* 0=uint16, 1=int16, 2=uint32, 3=int32, 4=float32 *)
    lrScale : LREAL := 1;
    lrOffset : LREAL;
    xHasSentinel : BOOL;
    dwSentinel : DWORD; (* Canonical bit order BEFORE scaling *)
END_VAR
VAR
    wA, wB, wTemporary : WORD;
    dwBits : DWORD;
    uBits : U_EmsReal32;
    lrRaw : LREAL;
END_VAR
(* IMPLEMENTATION *)
F_EmsDecode32.Valid := FALSE;
F_EmsDecode32.Value := 0;
wA := wFirst;
wB := wSecond;
IF xLowByteFirst THEN
    wA := SHL(wA AND WORD#16#00FF, 8) OR SHR(wA, 8);
    wB := SHL(wB AND WORD#16#00FF, 8) OR SHR(wB, 8);
END_IF;
IF xLowWordFirst AND (usiEncoding >= 2) THEN
    wTemporary := wA; wA := wB; wB := wTemporary;
END_IF;
IF usiEncoding < 2 THEN
    dwBits := WORD_TO_DWORD(wA);
ELSE
    dwBits := SHL(WORD_TO_DWORD(wA), 16) OR WORD_TO_DWORD(wB);
END_IF;
IF xHasSentinel AND (dwBits = dwSentinel) THEN RETURN; END_IF;
CASE usiEncoding OF
    0: lrRaw := WORD_TO_LREAL(wA);
    1:
        lrRaw := WORD_TO_LREAL(wA);
        IF wA >= WORD#16#8000 THEN lrRaw := lrRaw - LREAL#65536; END_IF;
    2: lrRaw := UDINT_TO_LREAL(DWORD_TO_UDINT(dwBits));
    3:
        lrRaw := UDINT_TO_LREAL(DWORD_TO_UDINT(dwBits));
        IF dwBits >= DWORD#16#80000000 THEN lrRaw := lrRaw - LREAL#4294967296; END_IF;
    4:
        IF (dwBits AND DWORD#16#7F800000) = DWORD#16#7F800000 THEN RETURN; END_IF; (* NaN/Inf *)
        uBits.Bits := dwBits;
        lrRaw := REAL_TO_LREAL(uBits.Value);
ELSE
    RETURN;
END_CASE;
F_EmsDecode32.Value := lrRaw * lrScale + lrOffset;
(* Practical engineering bound rejects NaN/overflow without target-specific math libraries. *)
F_EmsDecode32.Valid := (F_EmsDecode32.Value = F_EmsDecode32.Value)
    AND (ABS(F_EmsDecode32.Value) <= LREAL#1.0E30) AND (lrScale <> 0);
END_FUNCTION

(* ---- F_EmsDecode64.st ---- *)
(* POU: FUNCTION F_EmsDecode64. Exact UInt64 reconstruction; never pass via LREAL. *)
FUNCTION F_EmsDecode64 : ULINT
VAR_INPUT
    Words : ARRAY[0..3] OF WORD;
    xLowWordFirst : BOOL;
    xLowByteFirst : BOOL;
END_VAR
VAR
    i, j : INT;
    w : WORD;
END_VAR
(* IMPLEMENTATION *)
F_EmsDecode64 := 0;
FOR i := 0 TO 3 DO
    IF xLowWordFirst THEN j := 3 - i; ELSE j := i; END_IF;
    w := Words[j];
    IF xLowByteFirst THEN
        w := SHL(w AND WORD#16#00FF, 8) OR SHR(w, 8);
    END_IF;
    F_EmsDecode64 := SHL(F_EmsDecode64, 16) OR WORD_TO_ULINT(w);
END_FOR;
(* Validate the vendor's invalid sentinel before passing xValueValid to FB_EmsSample. *)
END_FUNCTION

(* ---- FB_EmsHighAlarm.st ---- *)
(* Create a FUNCTION_BLOCK POU. Declarations above, implementation below the divider.
   Requires the CODESYS Standard library (TON). Example settings are not safety limits.
   One instance per condition. Call every scan from ONE acquisition/alarm task.
   Acknowledgement belongs to Alarm Manager, never to this block. *)
FUNCTION_BLOCK FB_EmsHighAlarm
VAR_INPUT
    lrValue       : LREAL;
    xValid        : BOOL;        (* Good, fresh sample AND valid mapping *)
    lrHigh        : LREAL;
    lrReset       : LREAL;       (* Must be below lrHigh: hysteresis *)
    tRaiseDelay   : TIME := T#2s;
    tClearDelay   : TIME := T#5s;
END_VAR
VAR_OUTPUT
    xActive       : BOOL;        (* Digital alarm expression; never writable by HMI *)
    xInputFault   : BOOL;        (* Separate communication/measurement alarm *)
    xConfigFault  : BOOL;
END_VAR
VAR
    fbRaise       : TON;
    fbClear       : TON;
END_VAR
(* ---- Implementation ---- *)
xConfigFault := (lrReset >= lrHigh);
xInputFault := NOT xValid;
IF xInputFault OR xConfigFault THEN
    fbRaise(IN := FALSE, PT := tRaiseDelay);
    fbClear(IN := FALSE, PT := tClearDelay);
    (* Hold last known condition; unavailable data must not clear a fault. *)
ELSE
    fbRaise(IN := (NOT xActive) AND (lrValue >= lrHigh), PT := tRaiseDelay);
    fbClear(IN := xActive AND (lrValue <= lrReset), PT := tClearDelay);
    IF fbRaise.Q THEN
        xActive := TRUE;
    ELSIF fbClear.Q THEN
        xActive := FALSE;
    END_IF;
END_IF;
END_FUNCTION_BLOCK

(* ---- FB_EmsSample.st ---- *)
(* POU: FUNCTION_BLOCK FB_EmsSample. Declaration above the divider; implementation below it. *)
FUNCTION_BLOCK FB_EmsSample
VAR_INPUT
    xSupported : BOOL := TRUE;
    xEnabled : BOOL := TRUE;
    xNewSample : BOOL; (* One pulse per completed acquisition, NOT each PLC cycle. *)
    xReadError : BOOL; (* Failed transaction pulse; retained words are not new data. *)
    xValueValid : BOOL := TRUE;
    xClockValid : BOOL;
    uliUtcMs : ULINT;
    uliMonotonicMs : ULINT; (* LTIME_TO_ULINT(LTIME()) / ULINT#1000000 *)
    udiStaleAfterMs : UDINT := 5000;
END_VAR
VAR_OUTPUT
    Meta : ST_EmsMeta;
    xAccept : BOOL; (* Copy the decoded value only when TRUE. *)
END_VAR
VAR
    xSeen : BOOL;
    uliLastMs : ULINT;
END_VAR
(* IMPLEMENTATION *)
xAccept := FALSE;
IF NOT xSupported THEN
    Meta.Quality := 4; (* unsupported *)
    Meta.ObservedAtMs := 0;
    Meta.Sequence := 0;
    xSeen := FALSE;
ELSIF NOT xEnabled THEN
    Meta.Quality := 5; (* disabled; retain the last observation *)
ELSIF xReadError THEN
    Meta.Quality := 2; (* bad; preserve last observation time and value *)
ELSIF xNewSample THEN
    IF xValueValid THEN
        xAccept := TRUE;
        xSeen := TRUE;
        uliLastMs := uliMonotonicMs;
        IF xClockValid AND (uliUtcMs > 0) THEN
            Meta.Quality := 0;
            Meta.ObservedAtMs := uliUtcMs;
        ELSE
            Meta.Quality := 1; (* uncertain: no trustworthy UTC *)
            Meta.ObservedAtMs := 0;
        END_IF;
        IF Meta.Sequence = UDINT#4294967295 THEN
            Meta.Sequence := 1;
        ELSE
            Meta.Sequence := Meta.Sequence + 1;
        END_IF;
    ELSE
        Meta.Quality := 2; (* sentinel, range error or unmapped enum *)
    END_IF;
ELSIF xSeen THEN
    IF uliMonotonicMs < uliLastMs THEN
        Meta.Quality := 2; (* monotonic clock reset; wait for a new sample *)
    ELSIF (uliMonotonicMs - uliLastMs) > UDINT_TO_ULINT(udiStaleAfterMs) THEN
        Meta.Quality := 3; (* stale; UTC observation time stays unchanged *)
    END_IF;
END_IF;
END_FUNCTION_BLOCK

(* ---- PRG_EmsAlarms.st ---- *)
(* Reference only: wire these inputs to the completed Modbus acquisition result.
   xTemperatureValid must include freshness, device health, range and finite-value checks.
   Schedule this program cyclically. Choose limits/delays during commissioning. *)
PROGRAM PRG_EmsAlarms
VAR
    lrTemperatureC    : LREAL;
    xTemperatureValid: BOOL := FALSE;
    fbTemperature    : FB_EmsHighAlarm;
END_VAR
(* ---- Implementation ---- *)
fbTemperature(
    lrValue := lrTemperatureC,
    xValid := xTemperatureValid,
    lrHigh := 45.0,
    lrReset := 42.0,
    tRaiseDelay := T#2s,
    tClearDelay := T#5s
);
(* Alarm Manager / digital expressions:
   bess.temperature.high    := PRG_EmsAlarms.fbTemperature.xActive
   bess.temperature.invalid := PRG_EmsAlarms.fbTemperature.xInputFault
   bess.alarm.config        := PRG_EmsAlarms.fbTemperature.xConfigFault
   Define all three in an ACK_REP alarm class. Do not reset digital alarms on ACK.
   Alarm Manager owns occurrence state, timestamps, archive and acknowledgment.
   These expressions do NOT need individual OPC UA boolean tag subscriptions. *)
END_PROGRAM

(* ---- PRG_EmsExample.st ---- *)
(* POU: PROGRAM PRG_EmsExample. Map the Inputs through your completed Modbus request. *)
PROGRAM PRG_EmsExample
VAR
    (* Replace these driver-bound inputs; none are invented automatic CODESYS diagnostics. *)
    aBatteryWords : ARRAY[0..2] OF WORD;
    xBatteryDone : BOOL; (* one pulse for a successful complete response *)
    xBatteryError : BOOL;
    xUtcSynchronized : BOOL;
    uliUtcMs : ULINT; (* Fill from SysTimeRtcHighResGet + clock synchronization health. *)
    uliMonotonicMs : ULINT;
    powerSample : FB_EmsSample;
    socSample : FB_EmsSample;
    decoded : ST_EmsDecoded;
    lrSoc : LREAL;
END_VAR
(* IMPLEMENTATION *)
uliMonotonicMs := LTIME_TO_ULINT(LTIME()) / ULINT#1000000;
(* Example vendor: signed kW, positive charge. Convert ONCE to W, positive discharge. *)
decoded := F_EmsDecode32(wFirst := aBatteryWords[0], wSecond := aBatteryWords[1],
    xLowWordFirst := FALSE, xLowByteFirst := FALSE, usiEncoding := 3,
    lrScale := -1000, lrOffset := 0, xHasSentinel := TRUE, dwSentinel := DWORD#16#80000000);
powerSample(xNewSample := xBatteryDone, xReadError := xBatteryError,
    xValueValid := decoded.Valid AND (ABS(decoded.Value) <= LREAL#2000000),
    xClockValid := xUtcSynchronized, uliUtcMs := uliUtcMs,
    uliMonotonicMs := uliMonotonicMs, udiStaleAfterMs := 5000);
IF powerSample.xAccept THEN GVL_Ems.Battery.ac.activePower.Value := decoded.Value; END_IF;
GVL_Ems.Battery.ac.activePower.Meta := powerSample.Meta;

lrSoc := WORD_TO_LREAL(aBatteryWords[2]) * LREAL#0.1;
socSample(xNewSample := xBatteryDone, xReadError := xBatteryError,
    xValueValid := (aBatteryWords[2] <> WORD#16#FFFF) AND (lrSoc >= 0) AND (lrSoc <= 100),
    xClockValid := xUtcSynchronized, uliUtcMs := uliUtcMs,
    uliMonotonicMs := uliMonotonicMs, udiStaleAfterMs := 5000);
IF socSample.xAccept THEN GVL_Ems.Battery.battery.soc.Value := lrSoc; END_IF;
GVL_Ems.Battery.battery.soc.Meta := socSample.Meta;
(* Call in one acquisition task. Do not expose a partially updated struct as an atomic snapshot. *)
END_PROGRAM
